(*********************************** G.D S.p.A. - Technical Department ***********************************
============= PROGRAM INFO ============
FOLDER:             TBD
MACHINES INVOLVED:  TBD 

============= DESCRIPTION =============
csp machine declaration

============= REVISIONS ===============
Date		Version	 	Author      	Description             
----------	-------		------------  	--------------------------------------------
2019/04/05 	0000.00	 	M.Grasso		Creation of the PRG

**********************************************************************************************************)
(*$R process_ref := prc; $*)
PROGRAM csp_case_topRail
VAR
	
	prc:											process;
	prc_path:										STRING;
	
END_VAR

_read_var_input();

_object_manager();

IF NOT objects_running()
THEN
	RETURN;	
END_IF

_read_process_image();

_mode_manager();

_set_runtime_properties();

(********************************* BODY *********************************)
(************************************************************************)

_handle_messages();

_write_output();

ACTION _handle_messages:
;
END_ACTION

ACTION _handle_process_test:
;
END_ACTION

ACTION _mode_manager:
IF process_mode_req_is_pending(prc)
THEN
    process_apply_mode_req_first_step(prc);
    CASE process_get_mode(prc) OF
        MODE_TO_ABSENT:
			;
        MODE_TO_INACTIVE:
			;
        MODE_TO_TEST:
			;
        MODE_TO_OPERATIONAL:
			;
    END_CASE
    process_apply_mode_req_second_step(prc);
END_IF
END_ACTION

ACTION _object_manager:
IF objects_initialization()
THEN
	sub_process_init(
		object_name					:= 'csp_case_topRail.prc', 
		process						:= csp_case.prc, 
		CONVERSION_this				:= prc);
		
	prc_path 						:= process_get_path(prc);
END_IF

IF objects_running()
THEN
	process_cycle(prc);
END_IF
END_ACTION

ACTION _read_process_image:
;
END_ACTION

ACTION _read_var_input:
;
END_ACTION

ACTION _set_runtime_properties:
;
END_ACTION

ACTION _write_output:
;
END_ACTION

END_PROGRAM

(* stored: Version 1.1.0.1, ProductVersion 3.1.4022.12
   POU csp_case_topRail: Id {bba97ac3-cac6-482a-92cb-6991846523c1}, SpecialFunc None
   Action _handle_messages: Id {591ea2bc-7938-4ace-a55e-6fad4e6502f9}
   Action _handle_process_test: Id {022b7986-b249-4484-ae41-40405449402f}
   Action _mode_manager: Id {68c6971f-625b-4d33-95d5-e236e3640471}
   Action _object_manager: Id {ec20f9ec-1e4e-409f-a229-548fa1752ee8}
   Action _read_process_image: Id {7b63c8de-edb4-4131-adaa-77289bc56303}
   Action _read_var_input: Id {3445aac7-f057-413d-b88e-46097efd271c}
   Action _set_runtime_properties: Id {d0e19033-a05f-4c15-973e-bf64d88becb7}
   Action _write_output: Id {835a1be9-315b-4025-aaff-2ba2415cb409} *)
